TYPE IncrementalEncoderProcesses :
STRUCT
	///Enable the counter reset on the C pulse
	enableCounterResetC: Process;
	///Disable the counter reset on the C pulse
	disableCounterResetC: Process;
END_STRUCT
END_TYPE

(* stored: Version 1.1.0.1, ProductVersion 3.1.4019.2
   DUT IncrementalEncoderProcesses: Id {37cab044-911b-442b-8821-f7df37066649} *)
